FUNCTION_BLOCK acionamento (* Basic Function Block Type *)
  (* Standard: 61499-2 *)
  (* Version 0.0, 15/01/2026, Schneider Electric, Template *)
  PACKAGE Hidryco.HidrycoLib;
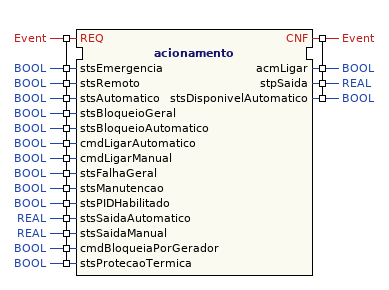
  EVENT_INPUT
    REQ WITH stsRemoto, stsAutomatico, stsBloqueioGeral, cmdLigarManual, cmdLigarAutomatico, stsBloqueioAutomatico, stsFalhaGeral, stsManutencao, stsPIDHabilitado, stsSaidaAutomatico, stsSaidaManual, cmdBloqueiaPorGerador, stsProtecaoTermica, stsEmergencia; (* Normal Execution Request *)
  END_EVENT
  EVENT_OUTPUT
    CNF WITH acmLigar, stpSaida, stsDisponivelAutomatico; (* Execution Confirmation *)
  END_EVENT
  VAR_INPUT
    stsEmergencia : BOOL;
    stsRemoto : BOOL;
    stsAutomatico : BOOL;
    stsBloqueioGeral : BOOL;
    stsBloqueioAutomatico : BOOL;
    cmdLigarAutomatico : BOOL;
    cmdLigarManual : BOOL;
    stsFalhaGeral : BOOL;
    stsManutencao : BOOL;
    stsPIDHabilitado : BOOL;
    stsSaidaAutomatico : REAL;
    stsSaidaManual : REAL;
    cmdBloqueiaPorGerador : BOOL;
    stsProtecaoTermica : BOOL;
  END_VAR
  VAR_OUTPUT
    acmLigar : BOOL;
    stpSaida : REAL;
    stsDisponivelAutomatico : BOOL; (* Status que o equipamento pode ser acionado em automatico *)
  END_VAR
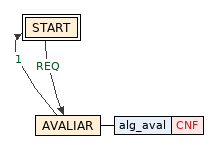
  EC_STATES
    START; (* Initial State *)
    AVALIAR : alg_aval -> CNF;
  END_STATES
  EC_TRANSITIONS
    START TO AVALIAR := REQ;
    AVALIAR TO START := 1;
  END_TRANSITIONS
  ALGORITHM alg_aval IN ST:
(* ============================================================
   CONTROLE DE ACIONAMENTO — Lógica principal
   ============================================================ *)

(* --- 1. Parada de emergência (prioridade máxima) --- *)
IF stsEmergencia THEN
    acmLigar := FALSE;
    stpSaida  := 0.0;
    RETURN;
END_IF;

(* --- 2. Condições de bloqueio geral --- *)
IF stsManutencao OR stsFalhaGeral OR NOT stsRemoto THEN
    acmLigar := FALSE;
    stpSaida  := 0.0;
    RETURN;
END_IF;

(* --- 3. Status de disponibilidade para modo automático --- *)
stsDisponivelAutomatico := stsAutomatico
                       AND NOT stsBloqueioAutomatico
                       AND NOT cmdBloqueiaPorGerador
                       AND NOT stsProtecaoTermica;

(* --- 4. Comando de ligar (automático ou manual) --- *)
IF stsAutomatico THEN
    acmLigar := cmdLigarAutomatico
            AND NOT stsBloqueioAutomatico
            AND NOT stsBloqueioGeral
            AND NOT cmdBloqueiaPorGerador
            AND NOT stsProtecaoTermica;
ELSE
    acmLigar := cmdLigarManual
            AND NOT stsBloqueioGeral
            AND NOT cmdBloqueiaPorGerador
            AND NOT stsProtecaoTermica;
END_IF;

(* --- 5. Seleção da fonte de saída --- *)
IF stsAutomatico AND stsPIDHabilitado THEN
    stpSaida := stsSaidaAutomatico;     (* PID ativo → saída automática *)
ELSE
    stpSaida := stsSaidaManual;         (* demais casos → saída manual  *)
END_IF;
;
  END_ALGORITHM
  ALGORITHM ALG_EMERGENCIA IN ST:
acmLigar := FALSE;
;
  END_ALGORITHM
END_FUNCTION_BLOCK
